Fanuc KAREL source: kb00121.KL

-- PROVISIONAL review KL for V1013-1; original PC SHA256 2b22c1f6f58a1df8a93292cef619fd0dd0056e9686eaf6307ee6c7931c5d32d9
-- Incomplete behavior may be omitted. Consult companion uncertainty JSON. Do not deploy.
PROGRAM KB00121
%NOLOCKGROUP
BEGIN
  -- UNRESOLVED_PC offsets 5-12; opcodes 9D,23
  -- UNRESOLVED_PC offsets 17-24; opcodes 9D,23
  -- UNRESOLVED_PC offsets 29-39; opcodes 9D,22,9D,33,35
  -- UNRESOLVED_PC offsets 44-51; opcodes 9D,23
  -- UNRESOLVED_PC offsets 56-90; opcodes 27,22,22,22,22,22,31
  -- UNRESOLVED_PC offsets 95-99; opcodes 7F
END KB00121
